// TwinCAT 3 PLC project use_axis
// ProgramVersion: 3.1.4023.0
// libraries:
//   Tc2_MC2, * (Beckhoff Automation GmbH)
//   Tc2_Standard, * (Beckhoff Automation GmbH)
//   Tc2_System, * (Beckhoff Automation GmbH)
//   Tc3_Module, * (Beckhoff Automation GmbH)
//   VisuDialogs, * (System)
// project tree:
//   DUTs/ E_MC_State.TcDUT, ST_HMI_Axis.TcDUT
//   / GlobalTextList.TcGTLO, PlcTask.TcTTO, Visualization Manager.TcVMO (not stored)
//   GVLs/ gHMI.TcGVL, gHW.TcGVL
//   POUs/ FB_axis.TcPOU, MAIN.TcPOU
//   VISUs/ main_tabs.TcVIS, vis_calibration.TcVIS, vis_motion.TcVIS
// real-time tasks:
//   TASK PlcTask: cycle T#10ms, priority 20, ADS port 350
// motion (NC):
//   TASK NC-Task 1 SAF: cycle T#2ms, priority 4, ADS port 501
//   TASK NC-Task 1 SVB: cycle T#10ms, priority 8, ADS port 511
//   AXIS Axis 1 (id 1)
//     General: UnitName=Degree
//     Dynamic: Acceleration=72000, Deceleration=72000, Jerk=216000
//     Velo: RefSearch=480, RefSync=480, SlowManual=2400, FastManual=14400, Fast=48000, Maximum=48000
//     OtherSettings: AllowMotionCmdToSlave=true, DataPersistence=true
//     encoder EncType=8
//       EncPara: ScaleFactorNumerator=360, ScaleFactorDenominator=1048576, Offset=-360.24787902832, MaxCount=#xffffffff, ReferenceSystem=1
//     drive DrvType=9
//       DrvPara: MaxCount=#xffffffff, DriveControlDWord=#x00030000
//         Analog: VeloReferenz=52800, VeloScale=1.02398817080127, TorqueScale=10, ScaleFactorActTorque=0.1
//         TimeComp: TaskDelayCycles=1
//     controller CtrType=1
//       CtrPara: PriorControlFactor=1
//         Observer: BandWidth=20
//   AXIS Axis 2 (id 2)
//     OtherSettings: AllowMotionCmdToSlave=true
//     encoder EncType=8
//       EncPara: MaxCount=#xffffffff
//     drive DrvType=9
//       DrvPara: MaxCount=#xffffffff, DriveControlDWord=#x00030000
//         Analog: VeloScale=1.02398817080127, TorqueScale=10, ScaleFactorActTorque=0.1
//         TimeComp: TaskDelayCycles=1
//     controller CtrType=1
//       CtrPara: PriorControlFactor=1
//         Observer: BandWidth=20
// I/O:
//   DEVICE Device 1 (EtherCAT), AmsNetId 5.19.209.26.2.1
//     Term 1 (EK1200) [EK1200-5000 EtherCAT Power supply (2A E-Bus)]
//       Term 2 (EL1094) [EL1094 4Ch. Dig. Input 24V, 10µs, negative]
//       Term 3 (EK1110) [EK1110 EtherCAT extension]
//     Drive 4 (AX5206-0000-0011) [AX5206-0000-0011 EtherCAT Drive (SoE, 2 Ch.)]
// variable links:
//   NC-Task 1 SAF/Axes/Axis 1 <-> Device 1 (EtherCAT)/Drive 4 (AX5206-0000-0011)
//     Drive/Inputs/In/nDcOutputTime <-> InfoData/DcOutputShift
//     Drive/Inputs/In/nState1 <-> AT 1/Drive status word @bit 8
//     Drive/Inputs/In/nState2 <-> AT 1/Drive status word
//     Drive/Inputs/In/nState4 @bit 1 <-> WcState/InputToggle
//     Drive/Inputs/In/nState4 <-> WcState/WcState
//     Drive/Outputs/Out/nCtrl1 <-> MDT 1/Master control word @bit 8
//     Drive/Outputs/Out/nDataOut2 <-> MDT 1/Velocity command value
//     Enc/Inputs/In/nDataIn1 <-> AT 1/Position feedback 1 value
//     Enc/Inputs/In/nDcInputTime <-> InfoData/DcInputShift
//     Enc/Inputs/In/nState4 @bit 1 <-> WcState/InputToggle
//     Enc/Inputs/In/nState4 <-> WcState/WcState
//   NC-Task 1 SAF/Axes/Axis 2 <-> Device 1 (EtherCAT)/Drive 4 (AX5206-0000-0011)
//     Drive/Inputs/In/nDcOutputTime <-> InfoData/DcOutputShift
//     Drive/Inputs/In/nState1 <-> AT 2/Drive status word @bit 8
//     Drive/Inputs/In/nState2 <-> AT 2/Drive status word
//     Drive/Inputs/In/nState4 @bit 1 <-> WcState/InputToggle
//     Drive/Inputs/In/nState4 <-> WcState/WcState
//     Drive/Outputs/Out/nCtrl1 <-> MDT 2/Master control word @bit 8
//     Drive/Outputs/Out/nDataOut2 <-> MDT 2/Velocity command value
//     Enc/Inputs/In/nDataIn1 <-> AT 2/Position feedback 1 value
//     Enc/Inputs/In/nDcInputTime <-> InfoData/DcInputShift
//     Enc/Inputs/In/nState4 @bit 1 <-> WcState/InputToggle
//     Enc/Inputs/In/nState4 <-> WcState/WcState
//   use_axis/use_axis Instance <-> NC-Task 1 SAF/Axes/Axis 1
//     PlcTask Inputs/MAIN.theAxis.NcToPlc <-> Outputs/ToPlc
//     PlcTask Outputs/MAIN.theAxis.PlcToNc <-> Inputs/FromPlc

CONFIGURATION use_axis
    RESOURCE PLC ON TwinCAT3
        TASK PlcTask(INTERVAL := T#10ms, PRIORITY := 20);
        PROGRAM MAIN WITH PlcTask : MAIN;
    END_RESOURCE
END_CONFIGURATION

// ---- DUTs/E_MC_State.TcDUT
TYPE E_MC_State :
(
	MCSTATE_Init,
	MCSTATE_NotPowered,
	MCSTATE_PowerOn,
	MCSTATE_PowerOff,
	MCSTATE_Idle,
	MCSTATE_Zero,
	MCSTATE_MoveAbs,
	MCSTATE_MoveRel,
	MCSTATE_MoveVel,
	MCSTATE_Jog,
	MCSTATE_Inch,
	MCSTATE_Home,
	MCSTATE_Stop,
	MCSTATE_Error,
	MCSTATE_Reset,
	MCSTATE_GearIn,
	MCSTATE_Geared,
	MCSTATE_GearOut,
	SaveBias
);

END_TYPE

// ---- DUTs/ST_HMI_Axis.TcDUT
TYPE ST_HMI_Axis :
STRUCT
	MoveRel: BOOL;
END_STRUCT
END_TYPE

// ---- GVLs/gHMI.TcGVL
{attribute 'qualified_only'}
VAR_GLOBAL
	AxisHMI_1: ST_HMI_Axis;
	bMoveRel : BOOL;
	bMoveAbs : BOOL;
	bMoveVel : BOOL;
	bMoveVel2 : BOOL;
	bStop : BOOL;
	vel 	: LREAL:=360;
	vel2 	: LREAL:=720;
	pos		: LREAL;
	targetAngle : LREAL;
	bias : LREAL;
	bSetHome : BOOL;
END_VAR

// ---- GVLs/gHW.TcGVL
{attribute 'qualified_only'}
VAR_GLOBAL
		//Axis: AXIS_REF;
END_VAR

// ---- POUs/MAIN.TcPOU
PROGRAM MAIN
VAR
	theAxis                  : AXIS_REF;
	fbAxis: FB_Axis;
	xState: E_MC_State;
	state : BYTE;	
	status : ST_AxisStatus;
	mcStatus : MC_ReadStatus;
	velo 	: LREAL;
	bRunVel	: BOOL;		
	mcReadParameter     : MC_ReadParameter;
END_VAR
VAR PERSISTENT
	str		  :	STRING(100):='This is a String';
	biasSaved : LREAL;
END_VAR

fbAxis(Axis:=theAxis);
theAxis.ReadStatus(); //HMI := gHMI.AxisHMI_1
//mcStatus(Axis := fbAxis.Axis, Enable := TRUE, Status=>status);
fbAxis.ReadPos(TRUE); gHMI.pos := fbAxis.actPos;
mcReadParameter(
		Axis:= theAxis, 
		Enable:= TRUE, 
		ParameterNumber:= MC_AxisParameter.AxisEncoderOffset, 
		ReadMode:= E_ReadMode.READMODE_ONCE
	);	
gHMI.bias := mcReadParameter.Value;
mcReadParameter(
		Axis:= theAxis, 
		Enable:= FALSE, 
		ParameterNumber:= MC_AxisParameter.AxisEncoderOffset, 
		ReadMode:= E_ReadMode.READMODE_ONCE
	);	

IF ABS(gHMI.bias - biasSaved) < 2 THEN
	str	:='Good: Home is calibrated!';
ELSE		
	str :='Warning: Home is NOT calibrated!';
END_IF
	
CASE xState OF
	MCSTATE_Init:		
		fbAxis.Enable(FALSE);		 
		IF theAxis.Status.Error THEN
			xState := MCSTATE_Error;
		ELSE	
			xState := MCSTATE_PowerOn;
		END_IF
		
	MCSTATE_PowerOn:
		fbAxis.Enable(TRUE);
		IF fbAxis.power.Done THEN
			//xState := MCSTATE_MoveRel;
			xState := MCSTATE_Idle;
		END_IF
		
	MCSTATE_Idle:		
		IF gHMI.bMoveRel THEN
			xState:= MCSTATE_MoveRel;
		END_IF	
		IF gHMI.bMoveAbs THEN
			xState:= MCSTATE_MoveAbs;
		END_IF									
		IF gHMI.bMoveVel THEN
			velo := gHMI.vel;		bRunVel := TRUE;			
			xState:= MCSTATE_MoveVel;  			
		END_IF
		IF gHMI.bMoveVel2 THEN
			velo := gHMI.vel2; 		bRunVel := TRUE;		
			xState:= MCSTATE_MoveVel; 				
		END_IF
		IF gHMI.bStop THEN
			xState:= MCSTATE_Stop;
		END_IF
		IF gHMI.bSetHome THEN
			xState:= SaveBias;
		END_IF
		
	MCSTATE_MoveVel:	
		fbAxis.MoveVel(bExecute := bRunVel, Velocity := velo, Direction := MC_Positive_Direction, 						
						acceleration := 1000, Deceleration := 1500, Jerk:= 0);	
		IF fbAxis.moveVels.Active OR fbAxis.moveVels.CommandAborted THEN
			bRunvel := FALSE; 				
		END_IF
		IF gHMI.bStop THEN
			xState:= MCSTATE_Stop;
			fbAxis.Stop(bExecute := FALSE, Deceleration := 1500, Jerk:= 0);					
		END_IF
		IF gHMI.bMoveVel THEN
			velo := gHMI.vel;			bRunvel := TRUE;						
		END_IF
		IF gHMI.bMoveVel2 THEN
			velo := gHMI.vel2;			bRunvel := TRUE;						
		END_IF
		
	MCSTATE_Stop:		
		fbAxis.Stop(bExecute := TRUE, Deceleration := 1500, Jerk:= 0);
		IF fbAxis.stops.Done  THEN
			fbAxis.Stop(bExecute := FALSE, Deceleration := 1500, Jerk:= 0);			
			xState := MCSTATE_Idle;
		END_IF
				
	MCSTATE_MoveRel:
		fbAxis.MoveRel(bExecute:=TRUE, relAngle:=360);		 
		IF fbAxis.moveRels.Done THEN
			fbAxis.MoveRel(bExecute:=FALSE, relAngle:=360);	
			xState :=  MCSTATE_Stop;
		END_IF
		
	MCSTATE_MoveAbs:
		fbAxis.MoveAbs(bExecute:=TRUE, targetAngle:=gHMI.targetAngle, velocityIncline:=720);		 
		IF fbAxis.moveAbses.Done THEN
			fbAxis.MoveAbs(bExecute:=FALSE, targetAngle:=gHMI.targetAngle, velocityIncline:=720);
			xState :=  MCSTATE_Stop;
		END_IF	
	
	SaveBias:		
		fbAxis.SaveBias();
		//gHMI.bias := fbAxis.lrPositionBias;			
		IF fbAxis.diState=0 THEN	
			//gHMI.bias := fbAxis.lrPositionBias;	
			biasSaved := fbAxis.lrPositionBias;		
			xState := MCSTATE_Init;		
		END_IF		
END_CASE

END_PROGRAM

// ---- POUs/FB_axis.TcPOU
FUNCTION_BLOCK FB_axis
VAR_INPUT
	//bStart							: BOOL;		
END_VAR
VAR_OUTPUT
	power	: ST_McOutputs;	
	resets	: ST_McOutputs;	
	estops	: ST_McOutputs;	
	stops	: ST_McOutputs;	
	driveResets	: ST_McOutputs;	
	diags		: ST_McOutputs;	
	diagNumber	: UDINT;
	moveRels  : ST_McOutputs;
	moveVels  : ST_McOutputs;
	moveAbses : ST_McOutputs;
	readVels	 : ST_McOutputs;
	actVel								: LREAL;
	readPoses	 : ST_McOutputs;
	actPos								: LREAL;
		lrPositionBias      : LREAL:=12321;
END_VAR
VAR_IN_OUT	
	Axis: AXIS_REF;
END_VAR
VAR	
	//eState		: axisState;
	mcPower		: MC_Power;
	mcReset		: MC_Reset;
	//mcDriveReset: FB_SoEReset;
	mcMoveAbs	: MC_MoveAbsolute;
	mcStop		: MC_Stop;
	mcMoveRel	: MC_MoveRelative;
	//mcReadDiag	: FB_SoEReadDiagNumber;
	mcReadVel	: MC_ReadActualVelocity;
	mcReadPos	: MC_ReadActualPosition;
	mcMoveVel	: MC_MoveVelocity;
	
	mcSetPos			: MC_SetPosition;
	mcReadParameter     : MC_ReadParameter;
    mcWritePersistent    : MC_WriteParameterPersistent;
	diState         	: DINT :=0;  // State machine variable
END_VAR

(*Axis.ReadStatus();

IF axis.Status.Error THEN
	eState := ERROR;	
END_IF
	

CASE eState OF
	INIT:
	           //gHW.errAck := TRUE; 
	    mcReset.Execute := FALSE;
		mcPower.Enable := FALSE;
		mcPower.Enable_Negative:= FALSE;
		mcPower.Enable_Positive:= FALSE;
		eState := ENABLE;
		
	ENABLE:		
	         //gHW.errAck := FALSE;
		mcPower.Enable := TRUE;
		mcPower.Enable_Negative:= TRUE;
		mcPower.Enable_Positive:= TRUE;
		IF mcPower.Status THEN
			eState := READY;
		END_IF	
		
	READY:
		IF bStart THEN
			eState:= ESTOP;
		END_IF
		
	ESTOP:		
		mcMoveRel.Distance := 100;
		mcMoveRel.Velocity := 100;
		mcMoveRel.Execute := TRUE;
		IF mcMoveRel.Done THEN
			mcMoveRel.Execute := FALSE;
			eState := READY;
		END_IF	
		
	ERROR:
		mcReset.Execute := TRUE;
		         //gHW.errAck := TRUE; 
		//mcPower.Enable := FALSE;
		//mcPower.Enable_Negative:= FALSE;
		//mcPower.Enable_Positive:= FALSE;
	    IF mcReset.Done THEN
			mcReset.Execute := FALSE;	
			eState := INIT;
		//eState := DISABLED;
		END_IF
END_CASE	

mcPower(Axis:= Axis);
mcMoveRel(Axis:= Axis);
mcReset(Axis:= Axis);*)

METHOD Enable : BOOL
VAR_INPUT
	bEnable : BOOL;
END_VAR
mcPower(
	Axis := Axis,
	Enable := bEnable,
	Enable_Positive := bEnable,
	Enable_Negative := bEnable,
	BufferMode := MC_Aborting,
	Override := 100,
	Status => power.Done,
	Error => power.Error
);
END_METHOD

METHOD eStop : BOOL
VAR_INPUT
	bExecute : BOOL;
END_VAR
VAR
	EStopDeceleration		: LREAL := 5000;
	EStopJerk				: LREAL := 20000;
END_VAR
mcStop(
	Axis := Axis,
	Execute := bExecute,
	Deceleration := EStopDeceleration,
	Jerk := EStopJerk,
	Done => estops.Done
);
END_METHOD

METHOD MoveAbs : BOOL
VAR_INPUT
	bExecute 			: BOOL;
	targetAngle 		: LREAL;
	velocityIncline		: LREAL;
END_VAR
VAR	
	accelerationIncline						: LREAL := 1000;
	decelerationIncline						: LREAL := 1500;
	jerkIncline								: LREAL;
END_VAR
mcMoveAbs(	
	Axis 		:= Axis,
	Execute 	:= bExecute,	
	Position			:= targetAngle,
	Velocity 			:= velocityIncline,//cali
	Acceleration 		:= accelerationIncline,
	Deceleration 		:= decelerationIncline,
	Jerk 				:= jerkIncline,	
	Done 			=> moveAbses.Done,
	Busy 			=> moveAbses.Busy,
	Active 			=> moveAbses.Active,
	CommandAborted 	=> moveAbses.CommandAborted,
	Error 			=> moveAbses.Error,
	ErrorID 		=> moveAbses.ErrorID,	
);
END_METHOD

METHOD MoveRel : BOOL
VAR_INPUT
	bExecute : BOOL;
	relAngle : LREAL;
END_VAR
VAR
	velocityIncline							: LREAL := 100;
	accelerationIncline						: LREAL := 1000;
	decelerationIncline						: LREAL := 1500;
	jerkIncline								: LREAL;
END_VAR
mcMoveRel(
	Axis := Axis,
	Execute := bExecute,
	Distance			:= relAngle,
	Velocity 			:= velocityIncline,//cali
	Acceleration 		:= accelerationIncline,
	Deceleration 		:= decelerationIncline,
	Jerk 				:= jerkIncline,	
	Done 			=> moveRels.Done,
	Busy 			=> moveRels.Busy,
	Active 			=> moveRels.Active,
	CommandAborted 	=> moveRels.CommandAborted,
	Error 			=> moveRels.Error,
	ErrorID 		=> moveRels.ErrorID
);
END_METHOD

METHOD MoveVel : BOOL
VAR_INPUT
	bExecute 		: BOOL;
	velocity		: LREAL;
	acceleration	: LREAL;
	deceleration	: LREAL;
	jerk			: LREAL;
	Direction		: MC_Direction;
END_VAR
VAR
	//BufferMode: MC_Aborting
END_VAR
mcMoveVel(	
	Axis 		:= Axis,
	Execute 	:= bExecute,		
	Velocity 			:= velocity*1,//speedCalibrationFactorL,//cali
	Acceleration 		:= acceleration,
	Deceleration 		:= deceleration,
	Jerk 				:= jerk,	
	BufferMode 			:= MC_Aborting,
	InVelocity 		=> moveVels.Done,
	Busy 			=> moveVels.Busy,
	Active 			=> moveVels.Active,
	CommandAborted 	=> moveVels.CommandAborted,
	Error 			=> moveVels.Error,
	ErrorID 		=> moveVels.ErrorID,	
);
END_METHOD

METHOD ReadMCparam : BOOL
VAR_INPUT
END_VAR
END_METHOD

METHOD ReadPos : BOOL
VAR_INPUT
	bEnable : BOOL;
END_VAR
mcReadPos (
	Axis := Axis,
	Enable := bEnable,
	Busy => readPoses.Busy,
	Position => ActPos
	//Error => diagNumberError,
	//AdsErrId => diagNumberAdsErrorID,
	//SercosErrId => diagNumberSercosErrorID 
);
END_METHOD

METHOD ReadVel : BOOL
VAR_INPUT
	bEnable : BOOL;
END_VAR
mcReadVel (
	Axis := Axis,
	Enable := bEnable,
	Busy => readVels.Busy,
	ActualVelocity => ActVel
	//Error => diagNumberError,
	//AdsErrId => diagNumberAdsErrorID,
	//SercosErrId => diagNumberSercosErrorID 
);
END_METHOD

METHOD Reset : BOOL
VAR_INPUT
	bExecute : BOOL;
END_VAR
mcReset(
	Axis := Axis,
	Execute := bExecute,
	Done => resets.Done,
	Error => resets.Error
);
END_METHOD

METHOD SaveBias : BOOL
VAR_INPUT
END_VAR
CASE diState OF	
  0:
  	diState := 5; // This step is required, 
				  // as we use 'diState=0' to determine that writing-persistent succeeds!    
  5:	
	mcSetPos(Axis:= Axis, Execute:=TRUE, Position :=0);
	IF NOT mcSetPos.Busy AND NOT mcSetPos.Error THEN
		mcSetPos(Axis:= Axis, Execute:= FALSE ); 
		diState := 10;           			
	END_IF
			
  10:
	mcReadParameter(
		Axis:= Axis, 
		Enable:= TRUE, 
		ParameterNumber:= MC_AxisParameter.AxisEncoderOffset, 
		ReadMode:= E_ReadMode.READMODE_ONCE
	);	
	IF NOT mcReadParameter.Busy AND NOT mcReadParameter.Error THEN       
		IF mcReadParameter.Valid THEN
			mcPower(Axis := Axis, Enable := FALSE,	Enable_Positive := FALSE,	Enable_Negative := FALSE);			
			//disable axis before writing-persistently!
			lrPositionBias := mcReadParameter.Value;
			diState := 0;//15;  	                 
		END_IF
		mcReadParameter(Axis:= Axis, Enable:= FALSE );
	END_IF
  15:
	diState := 20;  
	
  20: //write bias
	mcWritePersistent(Axis:= Axis, 
		Execute:= TRUE, ParameterNumber:= MC_AxisParameter.AxisEncoderOffset, Value:= lrPositionBias);  
		mcWritePersistent.ErrorID;
	IF NOT mcWritePersistent.Busy AND NOT mcWritePersistent.Error THEN
		mcWritePersistent(Axis:= Axis, Execute:= FALSE );
		diState     := 0;        
	END_IF		
END_CASE
END_METHOD

METHOD Stop : BOOL
VAR_INPUT
	bExecute : BOOL;
	Deceleration		: LREAL;
	Jerk				: LREAL;	
END_VAR
mcStop(
	Axis := Axis,
	Execute := bExecute,
	Deceleration := Deceleration,
	Jerk := Jerk,
	Done => stops.Done
);
END_METHOD

END_FUNCTION_BLOCK

// ---- GlobalTextList.TcGTLO
TEXTLIST GlobalTextList
  797 = '%.2f'
  288 = '%0.2f'
  228 = '%f'
  176 = '%s'
  532 = 'bias'
  543 = 'bias from Drive'
  488 = 'bias saved'
  798 = 'bias saved in Drive'
  554 = 'bias saved in PLC'
  221 = 'by Somebody'
  114 = 'Calibration'
  271 = 'Current Position'
  659 = 'Date'
  205 = 'Degree/s'
  377 = 'Motion'
  696 = 'Move Abs'
  403 = 'Move Relative'
  739 = 'Move Relative(360)'
  349 = 'Move To Angle:'
  687 = 'Move Velocity'
  105 = 'Move Velocity-1'
  280 = 'Move Velocity-2'
  528 = 'on Date'
  541 = 'Set Home'
  782 = 'Set Home / Save'
  173 = 'Stop'
  410 = 'targetAngle'
  260 = 'Velocity-1'
  921 = 'Velocity-2'
END_TEXTLIST

// ---- VISUs/main_tabs.TcVIS
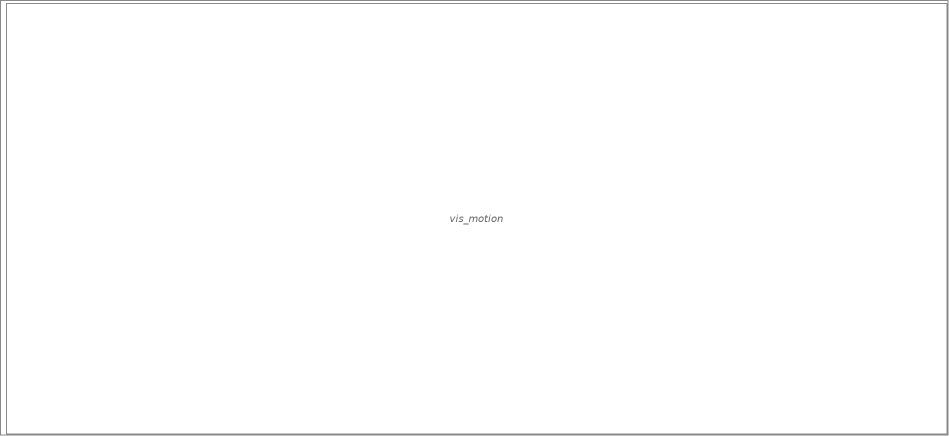
VISUALIZATION main_tabs  // 949x436
    TabControl (6,3 941x431)
        shows vis_motion()
        shows vis_calibration()
        [0]: TabTitle=Motion
        [1]: TabTitle=Calibration
END_VISUALIZATION

// ---- VISUs/vis_calibration.TcVIS
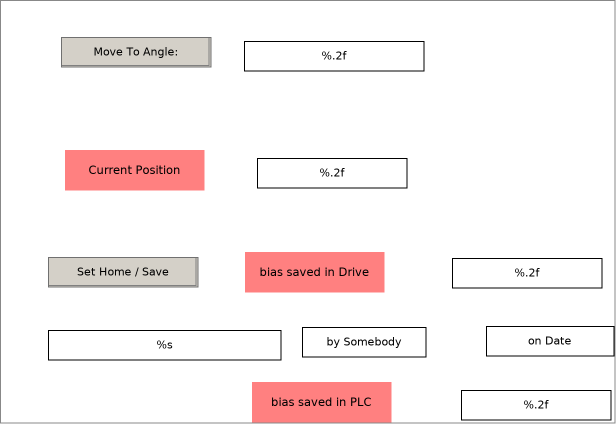
VISUALIZATION vis_calibration  // 616x424
    Rectangle (65,150 139x40), "Current Position"
    Button (61,37 150x30), "Move To Angle:"
        tap gHMI.bMoveAbs
    Rectangle (257,158 150x30), "%.2f", text variable: gHMI.pos
    Rectangle (244,41 180x30), "%.2f", text variable: gHMI.targetAngle
        OnMouseDown: write the text variable via Default
    Rectangle (245,252 139x40), "bias saved in Drive"
    Rectangle (452,258 150x30), "%.2f", text variable: gHMI.bias
    Button (48,257 150x30), "Set Home / Save"
        tap gHMI.bSetHome
    Rectangle (48,330 233x30), "%s", text variable: MAIN.str
        OnMouseDown: write the text variable via Default
    Rectangle (461,390 150x30), "%.2f", text variable: MAIN.biasSaved
    Rectangle (252,382 139x40), "bias saved in PLC"
    Rectangle (302,327 124x30), "by Somebody"
        OnMouseDown: write the text variable via Default
    Rectangle (486,326 128x30), "on Date"
        OnMouseDown: write the text variable via Default
END_VISUALIZATION

// ---- VISUs/vis_motion.TcVIS
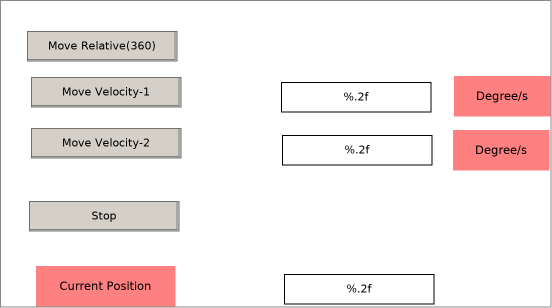
VISUALIZATION vis_motion  // 552x308
    Button (27,31 150x30), "Move Relative(360)"
        tap gHMI.bMoveRel
    Button (31,77 150x30), "Move Velocity-1"
        tap gHMI.bMoveVel
    Button (29,201 150x30), "Stop"
        tap gHMI.bStop
    Rectangle (453,130 96x40), "Degree/s"
    Rectangle (454,76 96x40), "Degree/s"
    Button (31,128 150x30), "Move Velocity-2"
        tap gHMI.bMoveVel2
    Rectangle (281,82 150x30), "%.2f", text variable: gHMI.vel
    Rectangle (282,135 150x30), "%.2f", text variable: gHMI.vel2
    Rectangle (36,266 139x40), "Current Position"
    Rectangle (284,274 150x30), "%.2f", text variable: gHMI.pos
END_VISUALIZATION
